PROGRAM P_FastTask
VAR
	
END_VAR

//MAIN.Serial1();
//MAIN.Serial2();
//MAIN.SerialRemoteFar(JoyStickNumber := GVL_HMI.unJoystick1SelectNum, Timeout := T#10S, ScreenActive => GVL_HMI.JoyStick1ScreenState);
//MAIN.SerialRemoteNear(JoyStickNumber := GVL_HMI.unJoystick2SelectNum, Timeout := T#10S, ScreenActive => GVL_HMI.JoyStick2ScreenState);

END_PROGRAM

(* stored: Version 1.1.0.1, ProductVersion 3.1.4022.3
   POU P_FastTask: Id {6857ec0c-81e9-416d-b00e-718270e310d9}, SpecialFunc None *)
